FUNCTION WithinTolerance : BOOL
VAR_INPUT
	value : LREAL;
	target : LREAL;
	tolerance : LREAL;
END_VAR
(*
checks if value is close enough to target within a given margin
*)

WithinTolerance := ABS(value-target) < tolerance;

END_FUNCTION

(* stored: Version 1.1.0.1, ProductVersion 3.1.4024.11
   POU WithinTolerance: Id {4e9ced49-a952-4cb0-b414-35672bc8309e}, SpecialFunc None *)
